// Implicitly generated code : DO NOT EDIT
FUNCTION CheckRangeSigned : DINT
VAR_INPUT
	value, lower, upper: DINT;
END_VAR

// Implicitly generated code : Only an Implementation suggestion
{noflow}
IF (value < lower) THEN
	CheckRangeSigned := lower;
ELSIF(value > upper) THEN
	CheckRangeSigned := upper;
ELSE
	CheckRangeSigned := value;
END_IF
{flow}

END_FUNCTION

(* stored: Version 1.1.0.1, ProductVersion 3.1.4024.11
   POU CheckRangeSigned: Id {25981379-f393-039d-3495-10f30c1a2a10}, SpecialFunc CheckRangeSigned *)
